Staubli VAL3: dateBase.dtx

public bool bCenterPoint = true
public bool bFrameTeach = true
public bool bPLC
public bool bToolTeach
public bool bWorTbMoving
public frame fWorkTable = {x=1460.596362, y=35.712914, z=-199.189903, rx=-0.117127, ry=-0.30554, rz=-53.750077, fatherId=world[0]}
public jointRx jHome = {j1=40.634782, j2=24.616214, j3=104.715258, j4=-108.662815, j5=68.5261, j6=132.709054}
public mdesc mGrindingSpd = {accel=70, decel=70, tmax=100, leave=0.5, reach=0.5}
public mdesc mNomSpeed = {accel=36, vel=60, decel=36, rmax=2000, tmax=100, blend=cartesian, leave=5, reach=5}
public num nPrdRadius = 100.111913
public tool tTCP = {x=1.417, y=48.029, z=261.326, rx=-28.407, ry=-42.029, rz=-19.448, fatherId=flange[0], ioLink=valve1}
